// No-op I_Comm implementation for tests. FB_Roof/FB_RoofMotor call Comm.Publish / Comm.PublishLog
// (via FB_EventLog) on error/state edges; a null (unassigned) I_Comm reference there would fault the
// PLC, so every FB_Roof test instance is given one of these instead of a real MQTT connection.
FUNCTION_BLOCK FB_NullComm IMPLEMENTS BROTLib.I_Comm
VAR
	// number of Publish/PublishLog calls seen, in case a test ever wants to assert an event fired
	nPublishCalls		: UDINT;
	nPublishLogCalls	: UDINT;
END_VAR

METHOD Publish : BOOL
VAR_INPUT
	domain			: STRING(255) := 'environment';
	location		: STRING(255) := 'roof';
	parameter		: STRING(255);
	value			: STRING(255);
END_VAR
VAR_OUTPUT
	published	: BOOL;
END_VAR
nPublishCalls := nPublishCalls + 1;
published := TRUE;
Publish := TRUE;
END_METHOD

METHOD PublishLog : BOOL
VAR_INPUT
	level		: STRING(255) := 'INFO';
	message		: STRING(255);
END_VAR
VAR_OUTPUT
	published	: BOOL;
END_VAR
nPublishLogCalls := nPublishLogCalls + 1;
published := TRUE;
PublishLog := TRUE;
END_METHOD

END_FUNCTION_BLOCK

(* stored: Version 1.1.0.1, ProductVersion 3.1.4024.15
   POU FB_NullComm: Id {78831305-3941-44e3-b3e0-2f7e7528e9d4}, SpecialFunc None
   Method Publish: Id {708d8db2-8eac-4a88-9ff6-cb72a2fc3822}
   Method PublishLog: Id {e9980b27-b480-4670-a4bd-74e6f77ee55b} *)
